Universal Robots PolyScope program: test2objects.urp

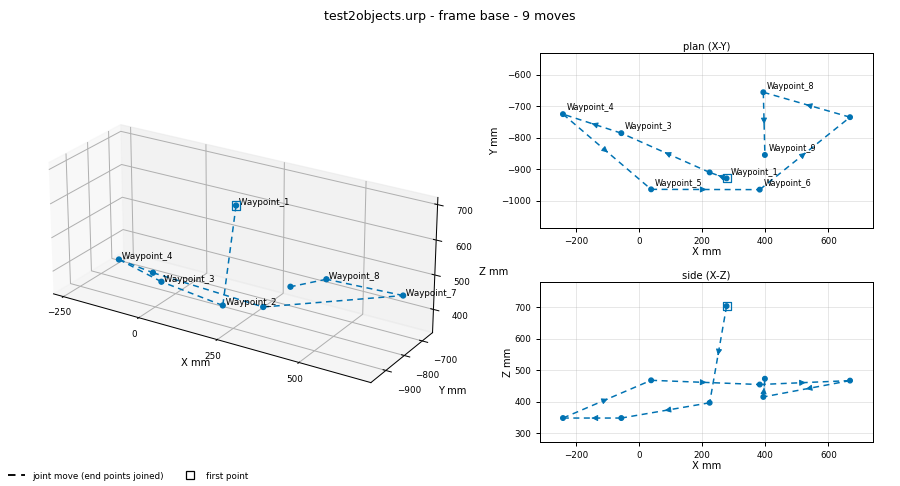
[picture p0: tool path of test2objects.urp in frame base, 9 of 9 moves have a stored position in this frame; points joined in program order, loops and branches not executed]
Program test2objects (installation=default directory=/programs/usbdisk/Test 2 createdIn=5.11.10.1010502 lastSavedIn=5.11.10.1010502 robotSerialNumber=20225201357)
Calibrated DH parameters: a=[-0.000097, -0.065329, -0.560646, 0.000001, -0.00004, 0]; d=[0.180831, -263.113709, 285.24385, -21.955837, 0.119737, 0.115719]; alpha=[1.571643, -0.002312, 0.004975, 1.569542, -1.570894, 0]; deltaTheta=[0, 1.463798, 5.013296, -0.193909, 0, 0]
Robot Program (runOnlyOnce=false)
  MoveJ speed 60 deg/s, acceleration 80 deg/s^2 (useActiveTCP=true) feature=Base
    Waypoint Waypoint_1: motionParameters(nextMotionTime=4); TCP in base x=277.402 y=-929.019 z=703.377 mm, rx=1.243 ry=0.9781 rz=-0.8768 rad; joints [93.191, -89.949, 87.689, 0.342, 85.312, 353.846] deg; TCP offset x=20.709 y=-1.468 z=254.962 mm, rx=-0.0022 ry=-0.0343 rz=-1.1076 rad
    Waypoint Waypoint_2: motionParameters(nextMotionTime=4); TCP in base x=223.741 y=-910.103 z=396.944 mm, rx=1.5671 ry=1.1083 rz=-0.8433 rad; joints [91.839, -85.257, 102.646, -1.132, 90.143, 353.804] deg
    Waypoint Waypoint_3: motionParameters(nextMotionTime=4); TCP in base x=-56.2 y=-785.722 z=348.517 mm, rx=1.605 ry=0.6842 rz=-1.2556 rad; joints [75.522, -97.039, 128.748, -29.315, 98.449, 353.643] deg
    Waypoint Waypoint_4: motionParameters(nextMotionTime=4); TCP in base x=-241.19 y=-725.409 z=348.54 mm, rx=1.605 ry=0.6842 rz=-1.2557 rad; joints [46.342, -102.609, 133.127, -28.02, 69.305, 352.411] deg
    Waypoint Waypoint_5: motionParameters(nextMotionTime=4); TCP in base x=38.202 y=-963.767 z=468.135 mm, rx=1.6076 ry=0.6612 rz=-1.2378 rad; joints [88.851, -82.985, 101.547, -16.109, 111.653, 355.686] deg
    Waypoint Waypoint_6: motionParameters(nextMotionTime=4); TCP in base x=382.468 y=-964.659 z=454.773 mm, rx=1.1833 ry=1.1303 rz=-0.6315 rad; joints [94.678, -79.525, 98.57, -16.103, 73.094, 355.662] deg
    Waypoint Waypoint_7: motionParameters(nextMotionTime=4); TCP in base x=668.699 y=-735.048 z=467.191 mm, rx=1.7559 ry=0.1517 rz=0.9615 rad; joints [115.757, -83.428, 103.57, -16.056, 73.112, 94.454] deg
    Waypoint Waypoint_8: motionParameters(nextMotionTime=4); TCP in base x=393.836 y=-656.015 z=415.462 mm, rx=1.7558 ry=0.1516 rz=0.9615 rad; joints [84.991, -103.026, 127.541, -18.782, 42.514, 91.382] deg
    Waypoint Waypoint_9: motionParameters(nextMotionTime=4); TCP in base x=398.814 y=-854.794 z=473.136 mm, rx=0.5419 ry=1.4424 rz=-0.0365 rad; joints [79.907, -73.477, 91.098, -20.588, 10.572, -4.348] deg
